FUNCTION_BLOCK FB_Lampe
VAR
    bOn : BOOL;
    bInit : BOOL := FALSE;
END_VAR

METHOD Init
VAR_INPUT
    fbManager : REFERENCE TO FB_Manager;
END_VAR
IF NOT bInit THEN
    fbManager.Register(THIS);
    bInit := TRUE;
END_IF
END_METHOD

END_FUNCTION_BLOCK

(* stored: Version 1.1.0.1
   POU FB_Lampe: Id {edafe033-5ac6-417f-a87d-e7aa768ed594}, SpecialFunc None
   Method Init: Id {cd5fdcba-8a5d-4724-ba83-73815cb7a11c} *)
